(* PLC project Tc2_Standard.R_TRIG Demo, tc3-libraries-kb TwinCAT 3.1 *)
(* stored: creationDateTime 2026-05-10T08:00:00, modificationDateTime 2026-05-10T08:00:00 *)

PROGRAM P_Demo_R_TRIG
  VAR
    fbR_TRIG : R_TRIG;  (* Trigger 实例 *)
    bButton : BOOL;  (* 按钮输入 *)
    bPress : BOOL;  (* 按钮按下沿（单周期脉冲） *)
  END_VAR

            // ============================================================
// Tc2_Standard.R_TRIG 演示程序
// ============================================================
// 场景：按钮按下（上升沿）时触发计数 +1
// 验证步骤：
//   1. 把本 PROGRAM 加到 PlcTask 调用列表
//   2. 编译并登录目标
//   1. bButton := FALSE 保持 → bPress 始终 FALSE
//   2. bButton := TRUE → bPress 在该周期为 TRUE，下一周期回 FALSE
//   3. bButton 持续 TRUE → bPress 不再触发，必须先 FALSE 再 TRUE
// ============================================================

fbR_TRIG(
    CLK := bButton,
    Q   => bPress
);

          
END_PROGRAM
